PROGRAM P_StringToConvExample
VAR
	s1	: STRING;
	s2	: STRING;
END_VAR

s1 := STRING_TO_CSVFIELD( 'Module_"ALFA_$05"_6', TRUE  );
s2 := STRING_TO_CSVFIELD( 'Module_50', FALSE );

s1 := CSVFIELD_TO_STRING( '"ab_$04_$05_cd-""ALFA""_5"', TRUE  );
s2 := CSVFIELD_TO_STRING( 'Module_50', FALSE );

END_PROGRAM

(* stored: Version 1.1.0.1, ProductVersion 3.1.4024.11
   POU P_StringToConvExample: Id {37f86ff5-868e-4575-9dde-a6497a03f5b5}, SpecialFunc None *)
